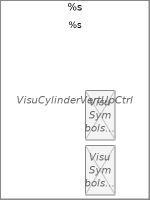
VISUALIZATION VisuCylinderVertUp  // 150x200
VAR_IN_OUT
	fbVisuCylinder: FB_VISU_CYLINDER;
END_VAR
    Image (85,90 30x50), invisible if: fbVisuCylinder.bWorkArrowInvisible, image: VisuSymbols.Symbols.ArrowBoldUp
        p2175578022: fbVisuCylinder.dwFrameColorWork
    Image (85,145 30x50), invisible if: fbVisuCylinder.bBaseArrowInvisible, image: VisuSymbols.Symbols.ArrowBoldDown
        p2175578022: fbVisuCylinder.dwFrameColorBase
    Group (25,90 40x100)
        p2738717112: fbVisuCylinder.iMove
        RoundedRectangle (10,0 20x100)
        RoundedRectangle (0,80 40x20)
    Rectangle (25,95 40x100)
        OnMouseClick: execute { fbVisuCylinder.bFrameInvisible:=false; }
    Textfield (0,15 150x20), "%s", text variable: fbVisuCylinder.strInfo, colour toggle: fbVisuCylinder.stEvent.bEventActive
    Textfield (0,0 150x14), "%s", text variable: fbVisuCylinder.strFullObjName
    Frame (0,0 150x200), invisible if: fbVisuCylinder.bFrameInvisible, frame switch variable: fbVisuCylinder.iFrame
        shows VisuCylinderVertUpCtrl(fbVisuCylinder := fbVisuCylinder)
END_VISUALIZATION

(* stored: Version 1.1.0.1, ProductVersion 3.1.4024.12
   Visu VisuCylinderVertUp: Id {665d85f4-e9d3-4b44-a48c-a32f8f7126fe} *)
